{attribute addProperty BoxType "EPP1111-0000-0016"}
{attribute addProperty Id "ID_InputsAT %I*ID_Inputs_90FEAF081620WcStateAT %I*WcState_98A4DF7520.250InfoDataAT %I*InfoData_BC63D37F80100"}
{attribute addProperty CRC "2402882033"}
{attribute addProperty SizeInBites "98"}
{attribute addProperty SizeInBytes "12.25"}
TYPE EPP1111_0792AF75 :
STRUCT
	{attribute addProperty Name "ID_Inputs"}
	ID_Inputs : ID_Inputs_90FEAF08;
	{attribute addProperty Name "WcState"}
	WcState : WcState_98A4DF75;
	{attribute addProperty Name "InfoData"}
	InfoData : InfoData_BC63D37F;
END_STRUCT
END_TYPE

(* stored: Version 1.2.0.0, ProductVersion 3.1.4024.9
   DUT EPP1111_0792AF75: Id {4e0bc562-122a-4db4-948c-e1e17e22b076} *)
